FUNCTION_BLOCK T_AddComponentCompareResultTrue EXTENDS T_UnitTestBase
VAR
  component1 : I_ComponentBase;
  list : T_ComponentsCollection;
  expected, actual : I_ComponentBase;
  result : BOOL;
END_VAR

list.AddComponent(component1);

result := expected = actual;
assertion.AssertEquals_BOOL(TRUE, result, 'result := expected = actual');
TestFinished();

END_FUNCTION_BLOCK

(* stored: Version 1.1.0.1, ProductVersion 3.1.4024.12
   POU T_AddComponentCompareResultTrue: Id {55b1b71c-5978-4695-ad7c-604fe3c44b7e}, SpecialFunc None *)
